PROGRAM MAIN
VAR
	PDUs:AllPDUs;
	CRAHs: AllCRAHs;
	IOStatus: All_IO;
	RTUStatus: AllRTUStat;
	CACs: AllCACs;
	IDF: AlllDF;
	OtherDIs: AllOtherDIs;
	EnergyMeters: AllEMeters;
	SystemTimeCall: SystemTime;
	ModbusComms: Modbus_RTU;
	
	bEmpryVar: BOOL;
	fTestFloat: REAL;
	bTestBool: BOOL;
	wTestWord: WORD;
END_VAR


ModbusComms();

CRAHs();
CACs();
PDUs();
IDF();
OtherDIs();
EnergyMeters();

IOStatus();
RTUStatus();

SystemTimeCall();

END_PROGRAM

(* stored: Version 1.1.0.1, ProductVersion 3.1.4024.12
   POU MAIN: Id {597f0add-bcb3-437c-8260-9c2a3e1283b3}, SpecialFunc None *)
